// Mitsubishi GX Works2 project: 1st   PLC: FX2N/FX2NC

PROGRAM MAIN
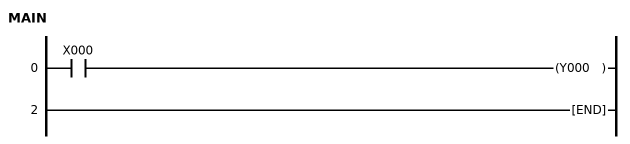
0     LD      X000
      OUT     Y000
2     END
END_PROGRAM
